// TIA Portal project "water tank control project" (V16)

(* hardware
DEVICE "S71500/ET200MP station_1"  S7-1500 station
   slot 0: "Rail_0"  Rack  6ES7 590-1***0-0AA0
   slot 1: "PLC_1"  CPU 1512C-1 PN  6ES7 512-1CK01-0AB0  V2.8
      slot 3: "CPU display_1"  6ES7591-1AA00-0AA0
      slot 32768: "PROFINET interface_1"  X1
         slot 32769: "Port_1"  X1 P1
         slot 32770: "Port_2"  X1 P2
      slot 34817: "Virtual CP interface port_1"  Virtual CP interface port  Virtual CP interface port
DEVICE "HMI_1"  TP900 Comfort
   slot 0: "HMI_1"  TP900 Comfort  6AV2 124-0JC01-0AX0  16.0.0.0
   slot 1: "HMI_RT_1"  TP900 Comfort  6AV2 124-0JC01-0AX0  16.0.0.0
   slot 5: "HMI_1.IE_CP_1"  PROFINET Interface  16.0.0.0
      slot 1: "PROFINET Interface_1"  PROFINET Interface
         slot 1: "Port_1"  Port
         slot 2: "Port_2"  Port
   slot 7: "HMI_1.MPI/DP_CP_1"  MPI/DP Interface  16.0.0.0
*)

// ===== PLC "PLC_1"  CPU 1512C-1 PN =====

VAR_GLOBAL   // PLC tag table "Default tag table"
   "set_reset_auto_1" AT %M4.0 : Bool;
   "s_r_manual" AT %M4.1 : Bool;
   "temp3" AT %M4.3 : Bool;
   "Clock_Byte" AT %MB0 : Byte;
   "Clock_10Hz" AT %M0.0 : Bool;
   "Clock_5Hz" AT %M0.1 : Bool;
   "Clock_2.5Hz" AT %M0.2 : Bool;
   "Clock_2Hz" AT %M0.3 : Bool;
   "Clock_1.25Hz" AT %M0.4 : Bool;
   "Clock_1Hz" AT %M0.5 : Bool;
   "Clock_0.625Hz" AT %M0.6 : Bool;
   "Clock_0.5Hz" AT %M0.7 : Bool;
END_VAR

VAR_GLOBAL   // PLC tag table "io"
   "AUTO" AT %I10.0 : Bool;
   "MANUAL" AT %I10.1 : Bool;
   "Start valve" AT %I10.2 : Bool;
   "stop valve" AT %I10.3 : Bool;
   "Start pump" AT %I10.4 : Bool;
   "Stop pump" AT %I10.5 : Bool;
   "STOP" AT %I10.6 : Bool;
   "WATER SENSOR" AT %IW0 : Int;
   "ValVE" AT %Q4.0 : Bool;
   "PUMP" AT %Q4.1 : Bool;
   "scaled output" AT %MD0 : Real;
   "hh_alarm_bool" AT %M1.0 : Bool;
   "LL_alarm_bool" AT %M1.1 : Bool;
   "error1_bit_bool" AT %M4.2 : Bool;
   "error1 (alarm)" AT %MW6 : Int;
END_VAR

DATA_BLOCK "HMI_connection"   // DB1
{ S7_Optimized_Access := 'TRUE' }
VERSION : 0.1
   VAR
      AUTO : Bool;
      manual : Bool;
      start_pump_PB : Bool;
      stop_pump_PB : Bool;
      start_valve_PB : Bool;
      stop_valve_PB : Bool;
      StOP_system_PB : Bool;
   END_VAR
   VAR RETAIN
      LOW_value_int : Int := 10;
      HIGH_value_int : Int := 50;
      time_before_start_valve : Time := T#5S;
      time_before_start_pump : Time := T#5S;
      LL_value_int : Int := 5;
      HH_value_int : Int := 55;
   END_VAR
BEGIN
END_DATA_BLOCK

DATA_BLOCK "auto_mode_DB"   // DB2
{ S7_Optimized_Access := 'TRUE' }
VERSION : 0.1
// stored: InstanceOfName auto_mode
"auto_mode"
BEGIN
END_DATA_BLOCK

DATA_BLOCK "manual_mode_DB"   // DB3
{ S7_Optimized_Access := 'TRUE' }
VERSION : 0.1
// stored: InstanceOfName manual_mode
"manual_mode"
BEGIN
END_DATA_BLOCK

DATA_BLOCK "alarms_DB"   // DB15
{ S7_Optimized_Access := 'TRUE' }
VERSION : 0.1
// stored: InstanceOfName alarms
"alarms"
BEGIN
END_DATA_BLOCK

DATA_BLOCK "errors_safety_DB"   // DB22
{ S7_Optimized_Access := 'TRUE' }
VERSION : 0.1
// stored: InstanceOfName errors_safety
"errors_safety"
BEGIN
END_DATA_BLOCK

// folder: System blocks/Program resources

DATA_BLOCK "IEC_Timer_0_DB"   // DB4
{ S7_Optimized_Access := 'TRUE' }
AUTHOR : Simatic
FAMILY : IEC
NAME : IEC_TMR
VERSION : 1.0
// stored: InstanceOfName IEC_TIMER
"IEC_TIMER"
BEGIN
END_DATA_BLOCK

DATA_BLOCK "IEC_Timer_0_DB_1"   // DB5
{ S7_Optimized_Access := 'TRUE' }
AUTHOR : Simatic
FAMILY : IEC
NAME : IEC_TMR
VERSION : 1.0
// stored: InstanceOfName IEC_TIMER
"IEC_TIMER"
BEGIN
END_DATA_BLOCK

DATA_BLOCK "time_before_start_empty"   // DB6
{ S7_Optimized_Access := 'TRUE' }
AUTHOR : Simatic
FAMILY : IEC
NAME : IEC_TMR
VERSION : 1.0
// stored: InstanceOfName IEC_TIMER
"IEC_TIMER"
BEGIN
END_DATA_BLOCK

DATA_BLOCK "IEC_Timer_0_DB_2"   // DB7
{ S7_Optimized_Access := 'TRUE' }
AUTHOR : Simatic
FAMILY : IEC
NAME : IEC_TMR
VERSION : 1.0
// stored: InstanceOfName IEC_TIMER
"IEC_TIMER"
BEGIN
END_DATA_BLOCK

DATA_BLOCK "IEC_Timer_0_DB_3"   // DB8
{ S7_Optimized_Access := 'TRUE' }
AUTHOR : Simatic
FAMILY : IEC
NAME : IEC_TMR
VERSION : 1.0
// stored: InstanceOfName IEC_TIMER
"IEC_TIMER"
BEGIN
END_DATA_BLOCK

DATA_BLOCK "IEC_Timer_0_DB_4"   // DB9
{ S7_Optimized_Access := 'TRUE' }
AUTHOR : Simatic
FAMILY : IEC
NAME : IEC_TMR
VERSION : 1.0
// stored: InstanceOfName IEC_TIMER
"IEC_TIMER"
BEGIN
END_DATA_BLOCK

DATA_BLOCK "IEC_Timer_0_DB_5"   // DB10
{ S7_Optimized_Access := 'TRUE' }
AUTHOR : Simatic
FAMILY : IEC
NAME : IEC_TMR
VERSION : 1.0
// stored: InstanceOfName IEC_TIMER
"IEC_TIMER"
BEGIN
END_DATA_BLOCK

DATA_BLOCK "IEC_Timer_0_DB_6"   // DB11
{ S7_Optimized_Access := 'TRUE' }
AUTHOR : Simatic
FAMILY : IEC
NAME : IEC_TMR
VERSION : 1.0
// stored: InstanceOfName IEC_TIMER
"IEC_TIMER"
BEGIN
END_DATA_BLOCK

DATA_BLOCK "IEC_Timer_0_DB_7"   // DB12
{ S7_Optimized_Access := 'TRUE' }
AUTHOR : Simatic
FAMILY : IEC
NAME : IEC_TMR
VERSION : 1.0
// stored: InstanceOfName IEC_TIMER
"IEC_TIMER"
BEGIN
END_DATA_BLOCK

DATA_BLOCK "IEC_Timer_0_DB_8"   // DB13
{ S7_Optimized_Access := 'TRUE' }
AUTHOR : Simatic
FAMILY : IEC
NAME : IEC_TMR
VERSION : 1.0
// stored: InstanceOfName IEC_TIMER
"IEC_TIMER"
BEGIN
END_DATA_BLOCK

DATA_BLOCK "IEC_Timer_0_DB_9"   // DB14
{ S7_Optimized_Access := 'TRUE' }
AUTHOR : Simatic
FAMILY : IEC
NAME : IEC_TMR
VERSION : 1.0
// stored: InstanceOfName IEC_TIMER
"IEC_TIMER"
BEGIN
END_DATA_BLOCK

DATA_BLOCK "IEC_Timer_0_DB_10"   // DB16
{ S7_Optimized_Access := 'TRUE' }
AUTHOR : Simatic
FAMILY : IEC
NAME : IEC_TMR
VERSION : 1.0
// stored: InstanceOfName IEC_TIMER
"IEC_TIMER"
BEGIN
END_DATA_BLOCK

DATA_BLOCK "IEC_Timer_0_DB_11"   // DB17
{ S7_Optimized_Access := 'TRUE' }
AUTHOR : Simatic
FAMILY : IEC
NAME : IEC_TMR
VERSION : 1.0
// stored: InstanceOfName IEC_TIMER
"IEC_TIMER"
BEGIN
END_DATA_BLOCK

DATA_BLOCK "IEC_Timer_0_DB_12"   // DB18
{ S7_Optimized_Access := 'TRUE' }
AUTHOR : Simatic
FAMILY : IEC
NAME : IEC_TMR
VERSION : 1.0
// stored: InstanceOfName IEC_TIMER
"IEC_TIMER"
BEGIN
END_DATA_BLOCK

DATA_BLOCK "IEC_Timer_0_DB_13"   // DB19
{ S7_Optimized_Access := 'TRUE' }
AUTHOR : Simatic
FAMILY : IEC
NAME : IEC_TMR
VERSION : 1.0
// stored: InstanceOfName IEC_TIMER
"IEC_TIMER"
BEGIN
END_DATA_BLOCK

DATA_BLOCK "IEC_Timer_0_DB_14"   // DB20
{ S7_Optimized_Access := 'TRUE' }
AUTHOR : Simatic
FAMILY : IEC
NAME : IEC_TMR
VERSION : 1.0
// stored: InstanceOfName IEC_TIMER
"IEC_TIMER"
BEGIN
END_DATA_BLOCK

DATA_BLOCK "IEC_Timer_0_DB_15"   // DB21
{ S7_Optimized_Access := 'TRUE' }
AUTHOR : Simatic
FAMILY : IEC
NAME : IEC_TMR
VERSION : 1.0
// stored: InstanceOfName IEC_TIMER
"IEC_TIMER"
BEGIN
END_DATA_BLOCK

// folder: (top level)

FUNCTION_BLOCK "auto_mode"   // FB1, LAD
{ S7_Optimized_Access := 'TRUE' }
VERSION : 0.1
   VAR_INPUT
      "water level" : Real;
      stop : Bool;
      LOW_value : Int;
      HIGH_value : Int;
   END_VAR
   VAR_IN_OUT
      "Pump out" : Bool;
      "valve out" : Bool;
   END_VAR
BEGIN

REGION Network 1: pump
   // default waiting time is 5s (it can be changet from HMI or from HMI_connecation_DB)
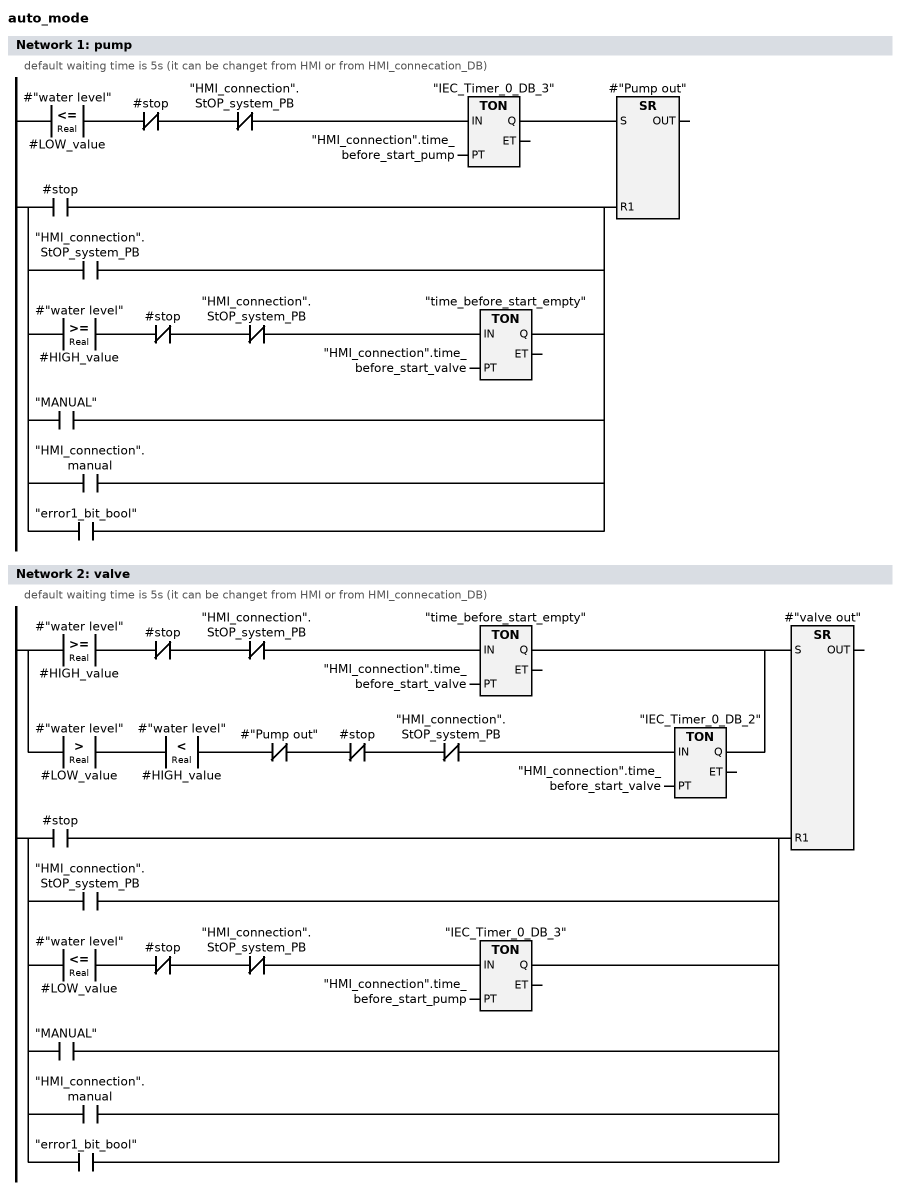
   "IEC_Timer_0_DB_3".TON(IN := (#"water level" <= #LOW_value) AND NOT #stop AND NOT "HMI_connection".StOP_system_PB,
                          PT := "HMI_connection".time_before_start_pump);
   "time_before_start_empty".TON(IN := (#"water level" >= #HIGH_value) AND NOT #stop AND NOT "HMI_connection".StOP_system_PB,
                           PT := "HMI_connection".time_before_start_valve);
   IF "IEC_Timer_0_DB_3".Q THEN
       #"Pump out" := TRUE;   // SR flip-flop
   END_IF;
   IF #stop OR "HMI_connection".StOP_system_PB OR "time_before_start_empty".Q OR "MANUAL" OR "HMI_connection".manual OR "error1_bit_bool" THEN
       #"Pump out" := FALSE;
   END_IF;
END_REGION

REGION Network 2: valve
   // default waiting time is 5s (it can be changet from HMI or from HMI_connecation_DB)
   "time_before_start_empty".TON(IN := (#"water level" >= #HIGH_value) AND NOT #stop AND NOT "HMI_connection".StOP_system_PB,
                           PT := "HMI_connection".time_before_start_valve);
   "IEC_Timer_0_DB_2".TON(IN := (#"water level" > #LOW_value) AND (#"water level" < #HIGH_value) AND NOT #"Pump out" AND NOT #stop AND NOT "HMI_connection".StOP_system_PB,
                          PT := "HMI_connection".time_before_start_valve);
   "IEC_Timer_0_DB_3".TON(IN := (#"water level" <= #LOW_value) AND NOT #stop AND NOT "HMI_connection".StOP_system_PB,
                          PT := "HMI_connection".time_before_start_pump);
   IF "time_before_start_empty".Q OR "IEC_Timer_0_DB_2".Q THEN
       #"valve out" := TRUE;   // SR flip-flop
   END_IF;
   IF #stop OR "HMI_connection".StOP_system_PB OR "IEC_Timer_0_DB_3".Q OR "MANUAL" OR "HMI_connection".manual OR "error1_bit_bool" THEN
       #"valve out" := FALSE;
   END_IF;
END_REGION
END_FUNCTION_BLOCK

FUNCTION_BLOCK "manual_mode"   // FB2, LAD
{ S7_Optimized_Access := 'TRUE' }
VERSION : 0.1
   VAR_INPUT
      "start valve PB" : Bool;
      "stop valve PB" : Bool;
      "stop system" : Bool;
      "start pump PB" : Bool;
      "stop pump PB" : Bool;
      HH_level : Int;
      LL_level : Int;
   END_VAR
   VAR_OUTPUT
      "pump output" : Bool;
      "valve output" : Bool;
   END_VAR
   VAR_IN_OUT
      "water level" : Real;
   END_VAR
BEGIN

REGION Network 1
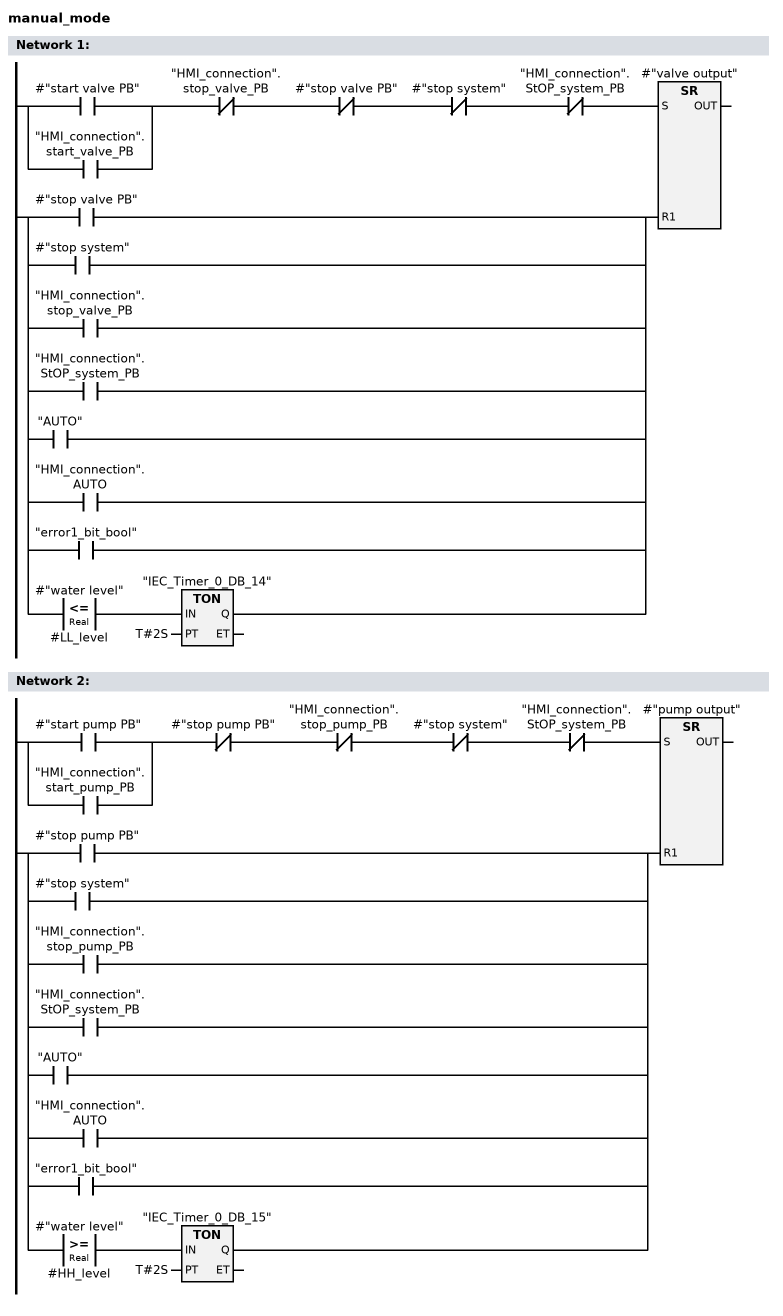
   "IEC_Timer_0_DB_14".TON(IN := #"water level" <= #LL_level, PT := T#2S);
   IF (#"start valve PB" OR "HMI_connection".start_valve_PB) AND NOT "HMI_connection".stop_valve_PB AND NOT #"stop valve PB" AND NOT #"stop system" AND NOT "HMI_connection".StOP_system_PB THEN
       #"valve output" := TRUE;   // SR flip-flop
   END_IF;
   IF #"stop valve PB" OR #"stop system" OR "HMI_connection".stop_valve_PB OR "HMI_connection".StOP_system_PB OR "AUTO" OR "HMI_connection".AUTO OR "error1_bit_bool" OR "IEC_Timer_0_DB_14".Q THEN
       #"valve output" := FALSE;
   END_IF;
END_REGION

REGION Network 2
   "IEC_Timer_0_DB_15".TON(IN := #"water level" >= #HH_level, PT := T#2S);
   IF (#"start pump PB" OR "HMI_connection".start_pump_PB) AND NOT #"stop pump PB" AND NOT "HMI_connection".stop_pump_PB AND NOT #"stop system" AND NOT "HMI_connection".StOP_system_PB THEN
       #"pump output" := TRUE;   // SR flip-flop
   END_IF;
   IF #"stop pump PB" OR #"stop system" OR "HMI_connection".stop_pump_PB OR "HMI_connection".StOP_system_PB OR "AUTO" OR "HMI_connection".AUTO OR "error1_bit_bool" OR "IEC_Timer_0_DB_15".Q THEN
       #"pump output" := FALSE;
   END_IF;
END_REGION
END_FUNCTION_BLOCK

FUNCTION_BLOCK "alarms"   // FB3, LAD
{ S7_Optimized_Access := 'TRUE' }
VERSION : 0.1
   VAR_INPUT
      LL_level : Int;
      HH_Level : Int;
      water_levle : Real;
   END_VAR
   VAR_OUTPUT
      HH_alarm : Bool;
      LL_alarm : Bool;
   END_VAR
BEGIN

REGION Network 1
   // hh
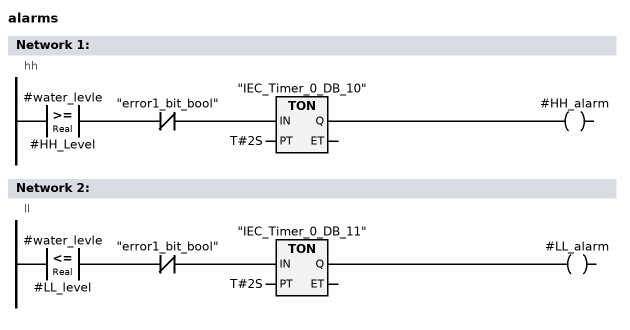
   "IEC_Timer_0_DB_10".TON(IN := (#water_levle >= #HH_Level) AND NOT "error1_bit_bool", PT := T#2S);
   #HH_alarm := "IEC_Timer_0_DB_10".Q;
END_REGION

REGION Network 2
   // ll
   "IEC_Timer_0_DB_11".TON(IN := (#water_levle <= #LL_level) AND NOT "error1_bit_bool", PT := T#2S);
   #LL_alarm := "IEC_Timer_0_DB_11".Q;
END_REGION
END_FUNCTION_BLOCK

FUNCTION_BLOCK "errors_safety"   // FB4, LAD
{ S7_Optimized_Access := 'TRUE' }
VERSION : 0.1
BEGIN

REGION Network 1: error 1
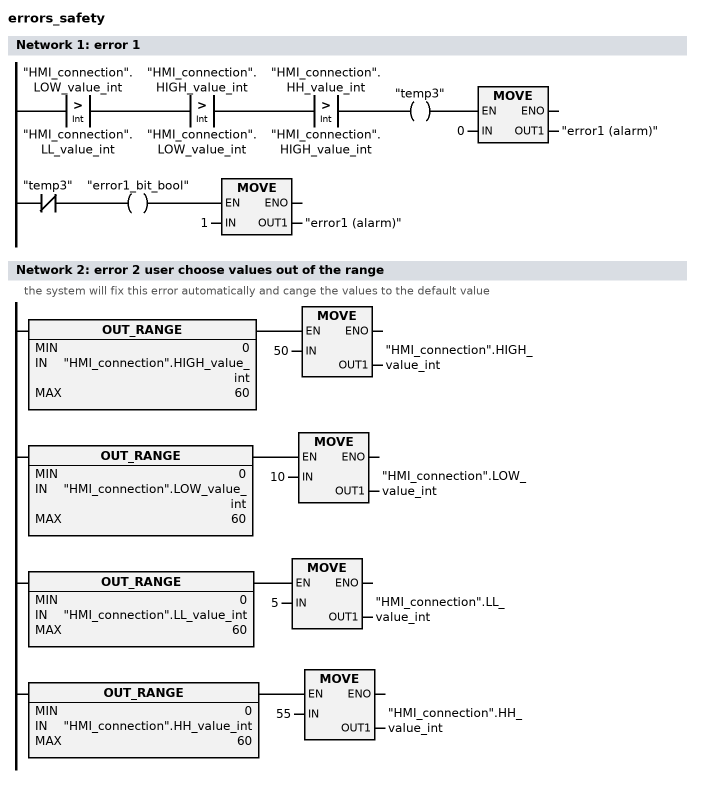
   RUNG wire#powerrail
      { S7_Templates := "SrcType := Int" } GT_Contact(in1 := "HMI_connection".LOW_value_int, in2 := "HMI_connection".LL_value_int)
      { S7_Templates := "SrcType := Int" } GT_Contact(in1 := "HMI_connection".HIGH_value_int, in2 := "HMI_connection".LOW_value_int)
      { S7_Templates := "SrcType := Int" } GT_Contact(in1 := "HMI_connection".HH_value_int, in2 := "HMI_connection".HIGH_value_int)
      Coil( "temp3" )
      Move(in := 0, out1 => "error1 (alarm)")
   END_RUNG
   RUNG wire#powerrail
      I_Contact( "temp3" )
      Coil( "error1_bit_bool" )
      Move(in := 1, out1 => "error1 (alarm)")
   END_RUNG
   // the same network as SCL:
   "temp3" := ("HMI_connection".LOW_value_int > "HMI_connection".LL_value_int) AND ("HMI_connection".HIGH_value_int > "HMI_connection".LOW_value_int) AND ("HMI_connection".HH_value_int > "HMI_connection".HIGH_value_int);
   IF "temp3" THEN "error1 (alarm)" := 0; END_IF;
   "error1_bit_bool" := NOT "temp3";
   IF NOT "temp3" THEN "error1 (alarm)" := 1; END_IF;
END_REGION

REGION Network 2: error 2 user choose values out of the range
   // the system will fix this error automatically and cange the values to the default value
   IF ("HMI_connection".HIGH_value_int < 0) OR ("HMI_connection".HIGH_value_int > 60) THEN
       "HMI_connection".HIGH_value_int := 50;
   END_IF;
   IF ("HMI_connection".LOW_value_int < 0) OR ("HMI_connection".LOW_value_int > 60) THEN
       "HMI_connection".LOW_value_int := 10;
   END_IF;
   IF ("HMI_connection".LL_value_int < 0) OR ("HMI_connection".LL_value_int > 60) THEN
       "HMI_connection".LL_value_int := 5;
   END_IF;
   IF ("HMI_connection".HH_value_int < 0) OR ("HMI_connection".HH_value_int > 60) THEN
       "HMI_connection".HH_value_int := 55;
   END_IF;
END_REGION
END_FUNCTION_BLOCK

FUNCTION "analogue set up" : Void   // FC1, LAD
{ S7_Optimized_Access := 'TRUE' }
VERSION : 0.1
   VAR_INPUT
      "Analogue inputs" : Int;
      LOWER : Int;
      HIGHER : Int;
   END_VAR
   VAR_OUTPUT
      "scaled output" : Real;
   END_VAR
   VAR_TEMP
      temp1 : Real;
   END_VAR
BEGIN

REGION Network 1
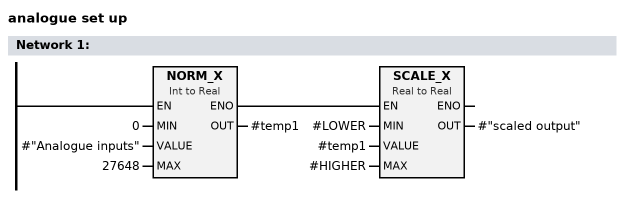
   RUNG wire#powerrail
      { S7_Templates := "[SrcType := Int, DestType := Real]" } Normalize(min := 0, value := #"Analogue inputs", max := 27648, out => #temp1)
      { S7_Templates := "[SrcType := Real, DestType := Real]" } Scale(min := #LOWER, value := #temp1, max := #HIGHER, out => #"scaled output")
   END_RUNG
   // the same network as SCL:
   #temp1 := NORM_X(MIN := 0, VALUE := #"Analogue inputs", MAX := 27648);
   #"scaled output" := SCALE_X(MIN := #LOWER, VALUE := #temp1, MAX := #HIGHER);
END_REGION
END_FUNCTION

ORGANIZATION_BLOCK "Main"   // OB1, LAD, ProgramCycle
TITLE = "Main Program Sweep (Cycle)"
{ S7_Optimized_Access := 'TRUE' }
VERSION : 0.1
   VAR_INPUT
      Initial_Call : Bool;   // Initial call of this OB
      Remanence : Bool;   // =True, if remanent data are available
   END_VAR
   VAR_TEMP
      set_reset_auto : Bool;
      set_reset_manual : Bool;
      temp1 : Int;
      tem2 : Bool;
      temp3 : Bool;
      temp4 : Bool;
   END_VAR
   VAR CONSTANT
      "LOW value" : Int := 10;
   END_VAR
BEGIN

REGION Network 1: analogue input set up
   // scaled output between 0-60 L
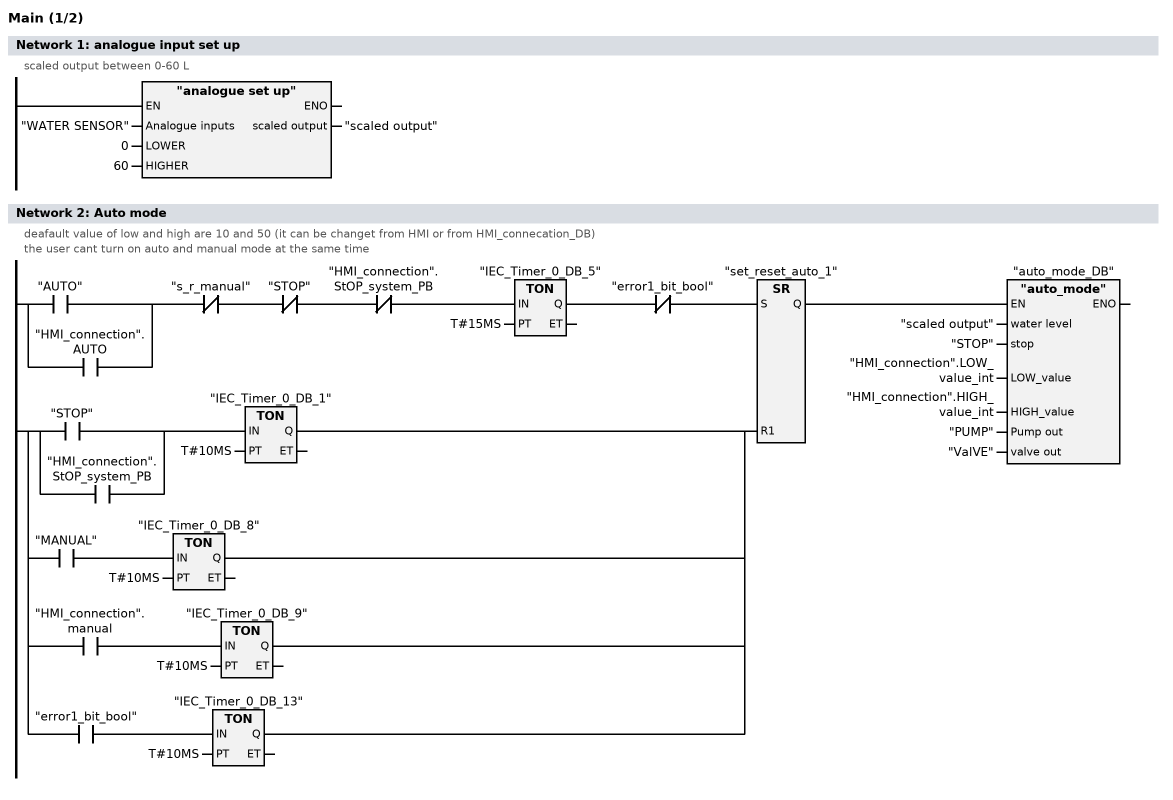
   RUNG wire#powerrail
      "analogue set up"("Analogue inputs" := "WATER SENSOR", LOWER := 0, HIGHER := 60, "scaled output" => "scaled output")
   END_RUNG
   // the same network as SCL:
   "analogue set up"("Analogue inputs" := "WATER SENSOR",
                     LOWER := 0,
                     HIGHER := 60,
                     "scaled output" => "scaled output");
END_REGION

REGION Network 2: Auto mode
   // deafault value of low and high are 10 and 50 (it can be changet from HMI or from HMI_connecation_DB)  
   // the user cant turn on auto and manual mode at the same time
   "IEC_Timer_0_DB_5".TON(IN := ("AUTO" OR "HMI_connection".AUTO) AND NOT "s_r_manual" AND NOT "STOP" AND NOT "HMI_connection".StOP_system_PB,
                          PT := T#15MS);
   "IEC_Timer_0_DB_1".TON(IN := "STOP" OR "HMI_connection".StOP_system_PB, PT := T#10MS);
   "IEC_Timer_0_DB_8".TON(IN := "MANUAL", PT := T#10MS);
   "IEC_Timer_0_DB_9".TON(IN := "HMI_connection".manual, PT := T#10MS);
   "IEC_Timer_0_DB_13".TON(IN := "error1_bit_bool", PT := T#10MS);
   IF "IEC_Timer_0_DB_5".Q AND NOT "error1_bit_bool" THEN
       "set_reset_auto_1" := TRUE;   // SR flip-flop
   END_IF;
   IF "IEC_Timer_0_DB_1".Q OR "IEC_Timer_0_DB_8".Q OR "IEC_Timer_0_DB_9".Q OR "IEC_Timer_0_DB_13".Q THEN
       "set_reset_auto_1" := FALSE;
   END_IF;
   IF "set_reset_auto_1" THEN
       "auto_mode_DB"("water level" := "scaled output",   // "auto_mode"
                      stop := "STOP",
                      LOW_value := "HMI_connection".LOW_value_int,
                      HIGH_value := "HMI_connection".HIGH_value_int,
                      "Pump out" := "PUMP",
                      "valve out" := "ValVE");
   END_IF;
END_REGION

REGION Network 3: manual mode
   // when we change to auto mode everything will be reset (pump valve)
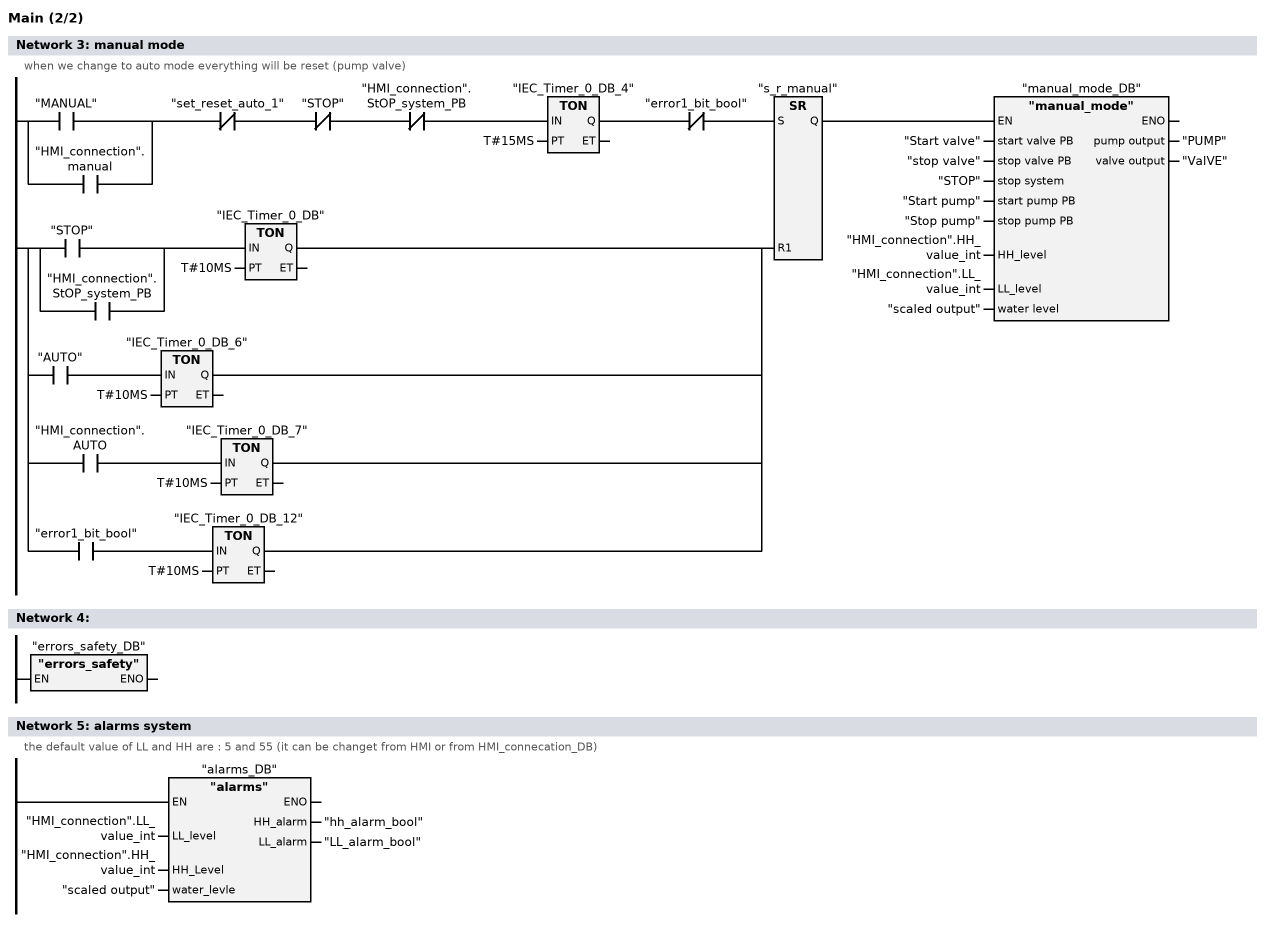
   "IEC_Timer_0_DB_4".TON(IN := ("MANUAL" OR "HMI_connection".manual) AND NOT "set_reset_auto_1" AND NOT "STOP" AND NOT "HMI_connection".StOP_system_PB,
                          PT := T#15MS);
   "IEC_Timer_0_DB".TON(IN := "STOP" OR "HMI_connection".StOP_system_PB, PT := T#10MS);
   "IEC_Timer_0_DB_6".TON(IN := "AUTO", PT := T#10MS);
   "IEC_Timer_0_DB_7".TON(IN := "HMI_connection".AUTO, PT := T#10MS);
   "IEC_Timer_0_DB_12".TON(IN := "error1_bit_bool", PT := T#10MS);
   IF "IEC_Timer_0_DB_4".Q AND NOT "error1_bit_bool" THEN
       "s_r_manual" := TRUE;   // SR flip-flop
   END_IF;
   IF "IEC_Timer_0_DB".Q OR "IEC_Timer_0_DB_6".Q OR "IEC_Timer_0_DB_7".Q OR "IEC_Timer_0_DB_12".Q THEN
       "s_r_manual" := FALSE;
   END_IF;
   IF "s_r_manual" THEN
       "manual_mode_DB"("start valve PB" := "Start valve",   // "manual_mode"
                        "stop valve PB" := "stop valve",
                        "stop system" := "STOP",
                        "start pump PB" := "Start pump",
                        "stop pump PB" := "Stop pump",
                        HH_level := "HMI_connection".HH_value_int,
                        LL_level := "HMI_connection".LL_value_int,
                        "water level" := "scaled output",
                        "pump output" => "PUMP",
                        "valve output" => "ValVE");
   END_IF;
END_REGION

REGION Network 4
   RUNG wire#powerrail
      "errors_safety_DB"()
   END_RUNG
   // the same network as SCL:
   "errors_safety_DB"();   // "errors_safety"
END_REGION

REGION Network 5: alarms system
   // the default value of LL and HH are : 5 and 55 (it can be changet from HMI or from HMI_connecation_DB)
   RUNG wire#powerrail
      "alarms_DB"(LL_level := "HMI_connection".LL_value_int, HH_Level := "HMI_connection".HH_value_int, water_levle := "scaled output", HH_alarm => "hh_alarm_bool", LL_alarm => "LL_alarm_bool")
   END_RUNG
   // the same network as SCL:
   "alarms_DB"(LL_level := "HMI_connection".LL_value_int,   // "alarms"
               HH_Level := "HMI_connection".HH_value_int,
               water_levle := "scaled output",
               HH_alarm => "hh_alarm_bool",
               LL_alarm => "LL_alarm_bool");
END_REGION
END_ORGANIZATION_BLOCK

(* ===== HMI "HMI_RT_1" =====
system functions are stored by id; their names below are inferred from use
connection "HMI_Connection_1": ETHERNET, S7_1500_OMS

HMI tags "Default tag table"
   "water_level.inp" : Real = PLC "scaled output" AT %MD0, 100 ms
   "valve.out" : Bool = PLC ValVE AT %Q4.0, 100 ms
   "pump.out" : Bool = PLC PUMP AT %Q4.1, 100 ms
   "AUTO" : Bool = PLC HMI_connection.AUTO AT %DB1.DBX0.0, 100 ms
   "MANUAL" : Bool = PLC HMI_connection.manual AT %DB1.DBX0.0, 100 ms
   "start_pump PB" : Bool = PLC HMI_connection.start_pump_PB AT %DB1.DBX0.0, 100 ms
   "stop_pump PB" : Bool = PLC HMI_connection.stop_pump_PB AT %DB1.DBX0.0, 100 ms
   "start_valve PB" : Bool = PLC HMI_connection.start_valve_PB AT %DB1.DBX0.0, 100 ms
   "stop_valve PB" : Bool = PLC HMI_connection.stop_valve_PB AT %DB1.DBX0.0, 100 ms
   "STOP_SYSTEM" : Bool = PLC HMI_connection.StOP_system_PB AT %DB1.DBX0.0, 100 ms
   "LOW_value" : Int = PLC HMI_connection.LOW_value_int AT %DB1.DBX0.0, 100 ms
   "HIGH_value" : Int = PLC HMI_connection.HIGH_value_int AT %DB1.DBW0, 100 ms
   "auto_mode_detector" : Bool = PLC set_reset_auto_1 AT %M4.0, 100 ms
   "manual_mode_detector" : Bool = PLC s_r_manual AT %M4.1, 100 ms
   "STOP_system_detector" : Bool AT %DB1.DBX0.0
   "time_before_start_valve" : Time = PLC HMI_connection.time_before_start_valve AT %DB1.DBD0, 100 ms
   "time_before_start_pump" : Time = PLC HMI_connection.time_before_start_pump AT %DB1.DBD0, 100 ms
   "HH_alarm_bool" : Bool = PLC hh_alarm_bool AT %M1.0, 100 ms
   "LL_alarm" : Bool = PLC LL_alarm_bool AT %M1.1, 100 ms
   "LL_value" : Int = PLC HMI_connection.LL_value_int AT %DB1.DBD0, 100 ms
   "HH_value" : Int = PLC HMI_connection.HH_value_int AT %DB1.DBW0, 100 ms
   "error1_bit (hh<h or LL>L)" : Bool = PLC error1_bit_bool AT %M4.2, 100 ms
   "erro1_bit_int_alarm" : Int = PLC "error1 (alarm)" AT %MW6, 100 ms

discrete alarms
   1: 'there is a inlogical choices that the user did in the values of the variabels', class Errors, trigger "erro1_bit_int_alarm" bit 0

analog alarms
   1: 'water level is too high', class Errors, trigger "water_level.inp"
   2: 'water level is too low', class Errors, trigger "water_level.inp"

screen "MAIN" 800x480
   SymbolLibrary "Symbol library_4" at 0,0 size 799x479
   Ellipse "Ellipse_1" at 661,276 size 96x113
      Appearance <- "valve.out"
   Circle "Circle_1" at 297,295 size 119x119
      Appearance <- "pump.out"
   SymbolLibrary "Template_Symbol library_3" at 626,360 size 65x11
   SymbolLibrary "Template_Symbol library_5" at 446,121 size 72x13
   SymbolLibrary "Template_Symbol library_4" at 488,78 size 146x311
   Bar "Template_Bar_1" at 512,90 size 93x298; Unit L; MinimumValue 0; MaximumValue 60
      ProcessValue <- "water_level.inp"
   SymbolLibrary "Template_Symbol library_2" at 690,293 size 39x79
   SymbolLibrary "Symbol library_1" at 419,121 size 28x25
   SymbolLibrary "Symbol library_2" at 419,140 size 15x198
   SymbolLibrary "Symbol library_3" at 404,337 size 30x26
   SymbolLibrary "Template_Symbol library_1" at 308,326 size 102x63
   SymbolLibrary "Template_Symbol library_6" at 729,360 size 70x11
   Button "Button_1" at 29,142 size 88x47; TextOff 'AUTO'
      on Press: function_b14e0dd5("AUTO", 0); ResetBit("STOP_system_detector")
      Appearance <- "auto_mode_detector"
   Button "Button_3" at 29,322 size 203x46; TextOff 'STOP'
      on Press: function_b14e0dd5("STOP_SYSTEM", 0); SetBit("STOP_system_detector")
      Appearance <- "STOP_system_detector"
   Button "Button_8" at 29,415 size 96x32; TextOff 'ALARMS'
      on Press: ActivateScreen("alarms", 0)
   Button "Button_9" at 133,415 size 96x32; TextOff 'VARIABELS'; Authorization "variabels"
      on Press: ActivateScreen("variabels", 0)
   Button "Button_2" at 141,142 size 88x47; TextOff 'MANUAL'
      on Press: function_b14e0dd5("MANUAL", 0); ResetBit("STOP_system_detector")
      Appearance <- "manual_mode_detector"
   Button "Button_4" at 29,201 size 88x47; TextOff 'start valve'
      on Press: function_b14e0dd5("start_valve PB", 0)
      Appearance <- "start_valve PB"
   Button "Button_5" at 141,201 size 88x47; TextOff 'start pump'
      on Press: function_b14e0dd5("start_pump PB", 0)
      Appearance <- "start_pump PB"
   Button "Button_6" at 31,262 size 88x47; TextOff 'stop valve'
      on Press: function_b14e0dd5("stop_valve PB", 0)
      Appearance <- "stop_valve PB"
   Button "Button_7" at 141,262 size 88x47; TextOff 'stop pump'
      on Press: function_b14e0dd5("stop_pump PB", 0)
      Appearance <- "stop_pump PB"
   IOField "I/O field_1" at 663,139 size 71x32; FormatPattern 99
      ProcessValue <- "LOW_value"
   IOField "I/O field_2" at 663,103 size 71x32; FormatPattern 99
      ProcessValue <- "HIGH_value"
   IOField "I/O field_3" at 663,185 size 71x32; FormatPattern 99
      ProcessValue <- "HH_value"
   IOField "I/O field_4" at 663,222 size 71x32; FormatPattern 99
      ProcessValue <- "LL_value"
   Circle "Circle_2" at 293,148 size 35x35
      Appearance <- "HH_alarm_bool"
   TextField "Text field_1" at 331,157 size 73x18; Text 'HH alarm'
   TextField "Text field_2" at 332,205 size 69x18; Text 'LL alarm'
   Circle "Circle_3" at 293,196 size 35x35
      Appearance <- "LL_alarm"
   TextField "Text field_3" at 692,109 size 13x20; Text 'L'
   TextField "Text field_4" at 692,145 size 13x20; Text 'L'
   TextField "Text field_5" at 692,191 size 13x20; Text 'L'
   TextField "Text field_6" at 692,227 size 13x20; Text 'L'
   TextField "Text field_7" at 733,108 size 57x18; Text 'H level'
   TextField "Text field_8" at 733,146 size 55x18; Text 'L level'
   TextField "Text field_10" at 733,228 size 63x18; Text 'LL level'
   TextField "Text field_11" at 733,194 size 67x18; Text 'HH level'
   Circle "Circle_4" at 293,241 size 35x35
      Appearance <- "error1_bit (hh<h or LL>L)"
   TextField "Text field_9" at 333,250 size 75x17; Text 'error 1 <>'

screen "alarms" 800x480
   SymbolLibrary "Symbol library_4" at 0,0 size 799x480
   AlarmView "Alarm view_1" at 0,0 size 800x415
   Button "Button_1" at 18,436 size 96x32; TextOff 'Back'
      on Press: function_efd93a16()

screen "variabels" 800x480
   SymbolLibrary "Symbol library_4" at 0,0 size 799x479
   IOField "I/O field_1" at 59,153 size 96x32; FormatPattern 99
      ProcessValue <- "LOW_value"
   IOField "I/O field_2" at 59,110 size 96x32; FormatPattern 99
      ProcessValue <- "HIGH_value"
   TextField "Text field_1" at 155,115 size 189x20; Text 'HIGH value of the water'
   TextField "Text field_2" at 155,161 size 186x20; Text 'LOW value of the water'
   IOField "I/O field_3" at 59,202 size 96x32; FormatPattern 99
      ProcessValue <- "LL_value"
   IOField "I/O field_4" at 59,243 size 96x32; FormatPattern 99
      ProcessValue <- "HH_value"
   TextField "Text field_3" at 156,207 size 338x20; Text 'LOW LOW level ( that will change the alarm)'
   TextField "Text field_4" at 156,247 size 339x20; Text 'HIGH HIGH level (that will change the alarm)'
   TextField "Text field_6" at 176,51 size 502x17; Text 'If the user inputs a value higher than the acceptable range (H=50/ HH=55)'
   TextField "Text field_5" at 159,21 size 565x22; Text 'The min and max values that the user should use are between 0-60'
   IOField "I/O field_5" at 59,292 size 96x32; FormatPattern 99999
      ProcessValue <- "time_before_start_valve"
   IOField "I/O field_6" at 60,336 size 96x32; FormatPattern 99999
      ProcessValue <- "time_before_start_pump"
   TextField "Text field_7" at 159,298 size 259x20; Text 'The pre-activation timer for valve'
   TextField "Text field_8" at 155,342 size 288x20; Text 'The pre-activation timer for the pump'
   Button "Button_1" at 22,428 size 96x32; TextOff 'Back'
      on Press: function_efd93a16()
   TextField "Text field_10" at 135,115 size 13x20; Text 'L'
   TextField "Text field_11" at 135,159 size 13x20; Text 'L'
   TextField "Text field_12" at 135,208 size 13x20; Text 'L'
   TextField "Text field_13" at 135,250 size 13x20; Text 'L'
   TextField "Text field_14" at 127,298 size 25x20; Text 'ms'
   TextField "Text field_15" at 127,342 size 25x20; Text 'ms'
   TextField "Text field_17" at 168,73 size 525x18; Text 'If the user inputs a value lower than the acceptable range (L=10/ LL=5)'
*)